// SIMATIC S7-200 project (STEP 7-Micro/WIN), CPU 214 REL 01.11

SYMBOL_TABLE DATOS
P1               I0.0     // PULSADOR 1
P2               I0.1     // PULSADOR 2
L                Q0.0     // LAMPARA
M1               M0.0     // TRANSICION 1
M2               M0.1     // TRANSICION 2
M3               M0.2     // TRANSICION 3
M4               M0.3     // TRANSICION 4
M5               M0.4     // TRANSICION 5
M6               M0.5     // TRANSICION 6
M7               M0.6     // TRANSICION 7
M8               M0.7     // TRANSICION 8
M9               M1.0     // TRANSICION 9
M10              M1.1     // TRANSICION 10
M11              M1.2     // TRANSICION 11
M12              M1.3     // TRANSICION 12
M13              M1.4     // TRANSICION 13
M14              M1.5     // TRANSICION 14
M15              M1.6     // TRANSICION 15
M16              M1.7     // TRANSICION 16
M17              M3.1     // TRANSICION 17
M18              M3.2     // TRANSICION 18
M19              M3.3     // TRANSICION 19
M20              M3.4     // TRANSICION 20
Q1               M2.0     // LUGAR 1
Q2               M2.1     // LUGAR 2
Q3               M2.2     // LUGAR 3
Q4               M2.3     // LUGAR 4
Q5               M2.4     // LUGAR 5
Q6               M2.5     // LUGAR 6
Q7               M2.6     // LUGAR 7
Q8               M2.7     // LUGAR 8
Q9               M3.0     // LUGAR 9
Q10              M3.5     // LUGAR 10
Q11              M3.6     // LUGAR 11
Q12              M3.7     // LUGAR 12
Q13              M4.0     // LUGAR 13
Ct2              T35      // TEMPORIZADOR DE 2 SEGUNDOS
END_SYMBOL_TABLE

ORGANIZATION_BLOCK PRINCIPAL:OB1
TITLE=COMENTARIOS DEL PROGRAMA
BEGIN
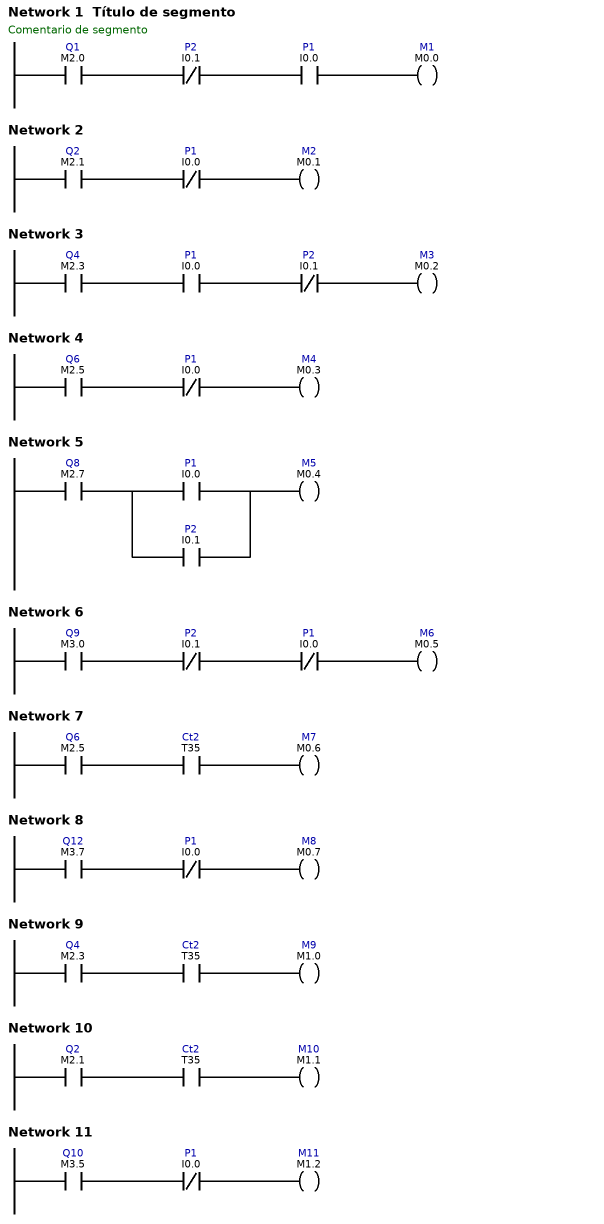
Network 1 // Título de segmento
// Comentario de segmento
LD     Q1:M2.0
AN     P2:I0.1
A      P1:I0.0
=      M1:M0.0
Network 2
// (network saved uncompiled; LAD cells follow)
// row 0: c0 -| |- Q2:M2.1  c1 -|/|- P1:I0.0  c2 -( ) M2:M0.1
Network 3
LD     Q4:M2.3
A      P1:I0.0
AN     P2:I0.1
=      M3:M0.2
Network 4
LD     Q6:M2.5
AN     P1:I0.0
=      M4:M0.3
Network 5
LD     Q8:M2.7
LD     P1:I0.0
O      P2:I0.1
ALD
=      M5:M0.4
Network 6
LD     Q9:M3.0
AN     P2:I0.1
AN     P1:I0.0
=      M6:M0.5
Network 7
LD     Q6:M2.5
A      Ct2:T35
=      M7:M0.6
Network 8
LD     Q12:M3.7
AN     P1:I0.0
=      M8:M0.7
Network 9
LD     Q4:M2.3
A      Ct2:T35
=      M9:M1.0
Network 10
LD     Q2:M2.1
A      Ct2:T35
=      M10:M1.1
Network 11
LD     Q10:M3.5
AN     P1:I0.0
=      M11:M1.2
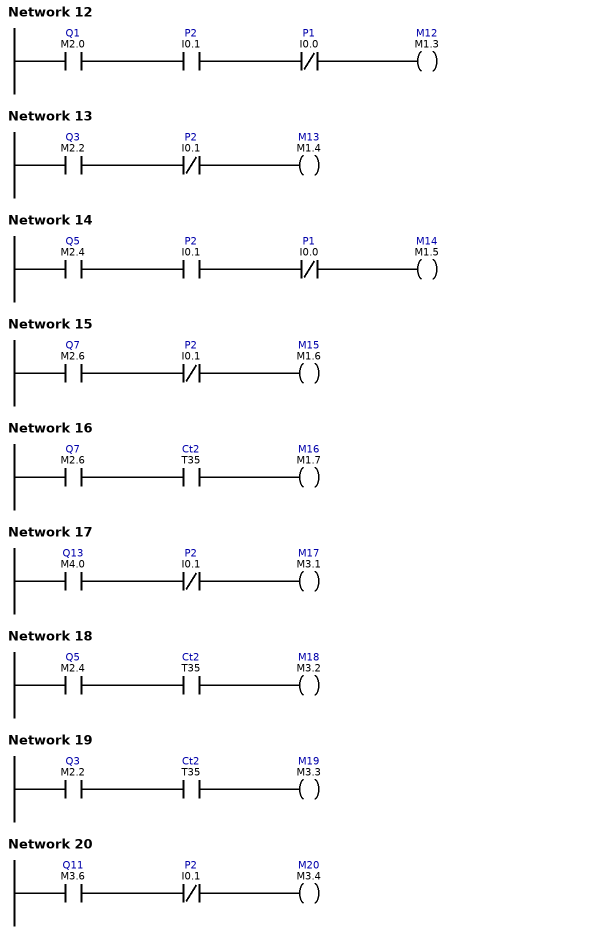
Network 12
LD     Q1:M2.0
A      P2:I0.1
AN     P1:I0.0
=      M12:M1.3
Network 13
LD     Q3:M2.2
AN     P2:I0.1
=      M13:M1.4
Network 14
LD     Q5:M2.4
A      P2:I0.1
AN     P1:I0.0
=      M14:M1.5
Network 15
LD     Q7:M2.6
AN     P2:I0.1
=      M15:M1.6
Network 16
LD     Q7:M2.6
A      Ct2:T35
=      M16:M1.7
Network 17
LD     Q13:M4.0
AN     P2:I0.1
=      M17:M3.1
Network 18
LD     Q5:M2.4
A      Ct2:T35
=      M18:M3.2
Network 19
LD     Q3:M2.2
A      Ct2:T35
=      M19:M3.3
Network 20
LD     Q11:M3.6
AN     P2:I0.1
=      M20:M3.4
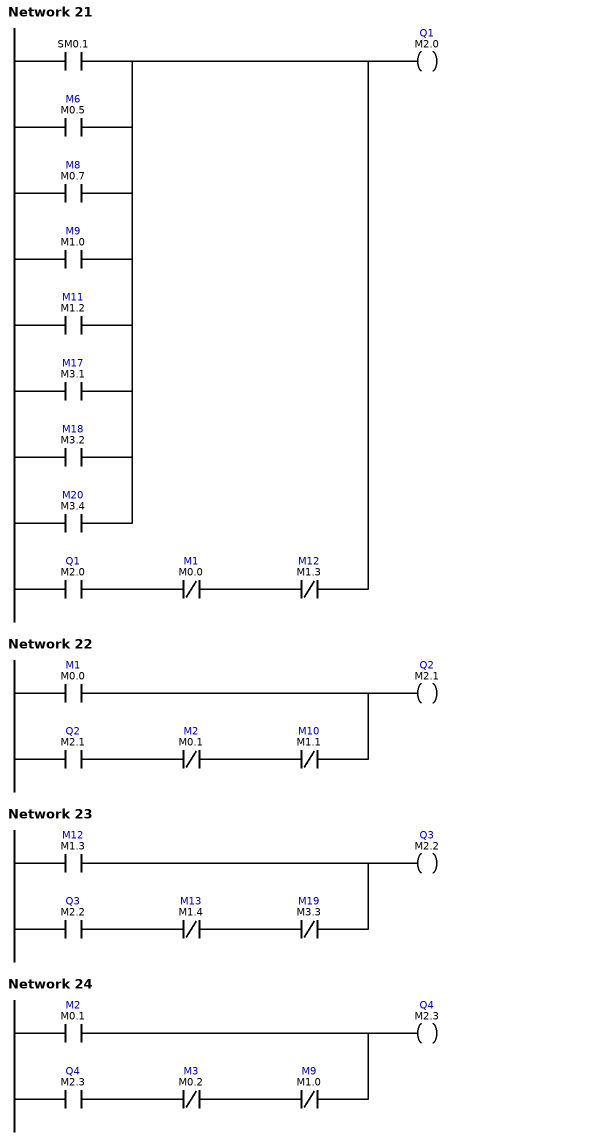
Network 21
LD     SM0.1
O      M6:M0.5
O      M8:M0.7
O      M9:M1.0
O      M11:M1.2
O      M17:M3.1
O      M18:M3.2
O      M20:M3.4
LD     Q1:M2.0
AN     M1:M0.0
AN     M12:M1.3
OLD
=      Q1:M2.0
Network 22
LD     M1:M0.0
LD     Q2:M2.1
AN     M2:M0.1
AN     M10:M1.1
OLD
=      Q2:M2.1
Network 23
LD     M12:M1.3
LD     Q3:M2.2
AN     M13:M1.4
AN     M19:M3.3
OLD
=      Q3:M2.2
Network 24
LD     M2:M0.1
LD     Q4:M2.3
AN     M3:M0.2
AN     M9:M1.0
OLD
=      Q4:M2.3
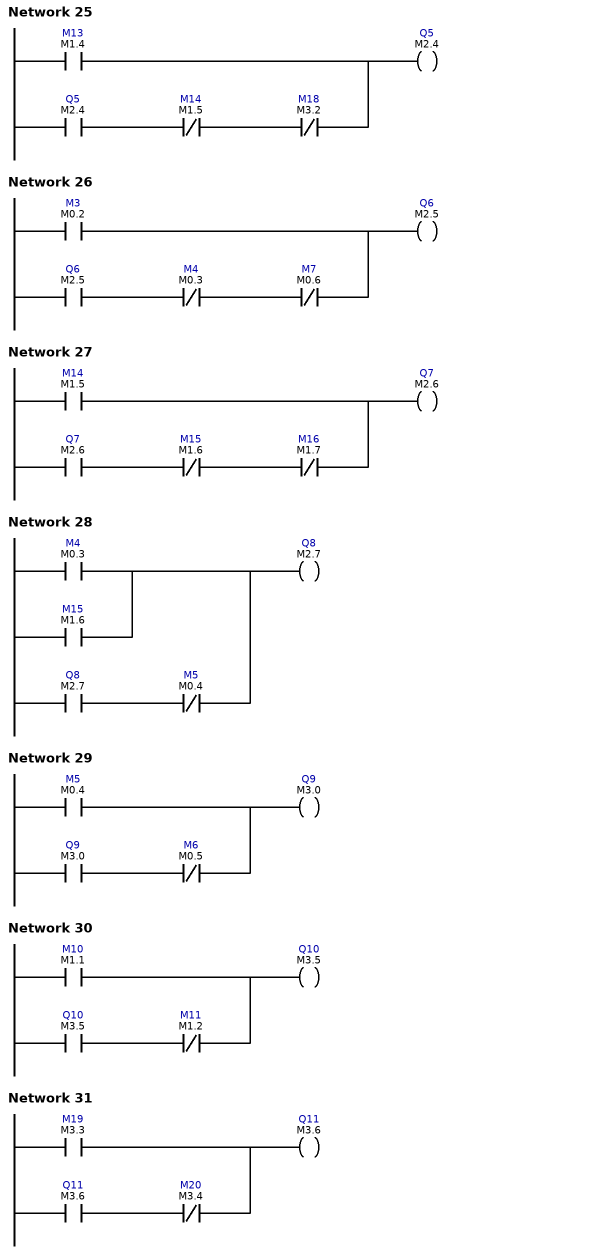
Network 25
LD     M13:M1.4
LD     Q5:M2.4
AN     M14:M1.5
AN     M18:M3.2
OLD
=      Q5:M2.4
Network 26
LD     M3:M0.2
LD     Q6:M2.5
AN     M4:M0.3
AN     M7:M0.6
OLD
=      Q6:M2.5
Network 27
LD     M14:M1.5
LD     Q7:M2.6
AN     M15:M1.6
AN     M16:M1.7
OLD
=      Q7:M2.6
Network 28
LD     M4:M0.3
O      M15:M1.6
LD     Q8:M2.7
AN     M5:M0.4
OLD
=      Q8:M2.7
Network 29
LD     M5:M0.4
LD     Q9:M3.0
AN     M6:M0.5
OLD
=      Q9:M3.0
Network 30
LD     M10:M1.1
LD     Q10:M3.5
AN     M11:M1.2
OLD
=      Q10:M3.5
Network 31
LD     M19:M3.3
LD     Q11:M3.6
AN     M20:M3.4
OLD
=      Q11:M3.6
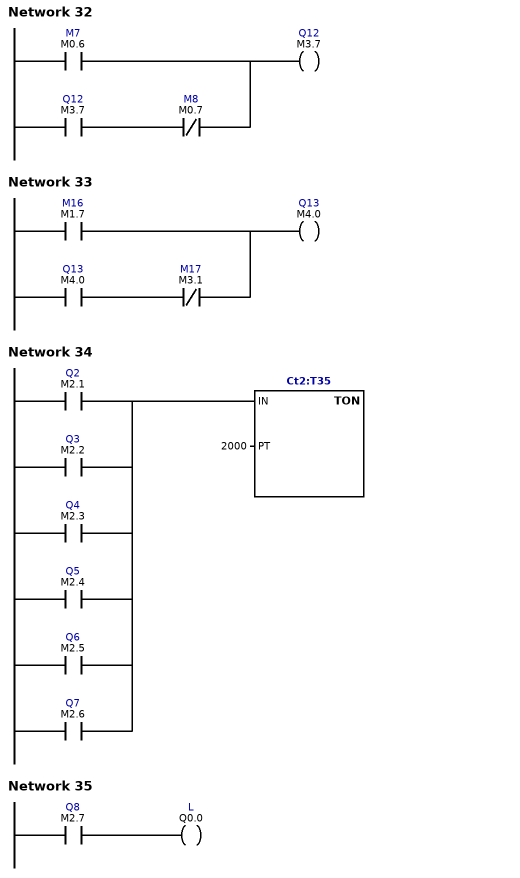
Network 32
LD     M7:M0.6
LD     Q12:M3.7
AN     M8:M0.7
OLD
=      Q12:M3.7
Network 33
LD     M16:M1.7
LD     Q13:M4.0
AN     M17:M3.1
OLD
=      Q13:M4.0
Network 34
LD     Q2:M2.1
O      Q3:M2.2
O      Q4:M2.3
O      Q5:M2.4
O      Q6:M2.5
O      Q7:M2.6
TON    Ct2:T35, 2000
Network 35
LD     Q8:M2.7
=      L:Q0.0
END_ORGANIZATION_BLOCK
